Yaskawa INFORM job: OK_R2_O22-23(-90,180)OKKR.JBI

/JOB
//NAME OK_R2_O22-23(-90,180)OKKR
///FOLDERNAME X4
//POS
///NPOS 107,107,107,5,0,0
///TOOL 0
///POSTYPE PULSE
///PULSE
C00000=-79400,-96450,-73119,-47071,38510,50576
C00001=-120689,-37236,-43262,-1430,36977,65337
C00002=-120661,8390,6118,-1752,30038,65509
C00003=-121363,14227,14389,-901,27936,65072
C00004=-121630,18134,20803,-569,25994,64899
C00005=-122051,20456,22985,52,25844,64579
C00006=-122335,22651,22887,-209,31352,64420
C00007=-122335,23153,24532,-213,30597,64422
C00008=-122573,22007,22272,73,31399,64269
C00009=-118553,33336,34533,32200,31167,63632
C00010=-118554,33797,35647,32601,30785,63423
C00011=-118795,35881,37778,33055,30674,63177
C00012=-119029,34698,36884,33342,30719,63021
C00013=-119029,35470,39068,34241,29924,62556
C00014=-119029,34698,36884,33342,30719,63021
C00015=-122566,16275,19454,818,25870,64189
C00016=-120682,5973,-10666,26006,48512,34380
C00017=-120682,6077,-8041,26626,47105,33962
C00018=-120965,19546,-3322,22995,60520,37308
C00019=-120686,6056,-8291,26571,47234,33999
C00020=-120521,4024,-8795,26757,46523,33864
C00021=-122243,21545,4650,37838,56763,29509
C00022=-115724,34900,14421,35017,60862,31707
C00023=-122685,12952,-4874,39297,55027,28576
C00024=-131885,-4518,-22891,42927,60902,26587
C00025=-120689,-37236,-43262,-1430,36977,65337
C00026=-79400,-96450,-73119,-47071,38510,50576
C00027=8645,-72931,-67050,-57733,95594,74029
C00028=3643,-76224,-106676,19950,71810,76872
C00029=266,-73751,-67438,-57600,90404,72524
C00030=-56065,-40103,-98025,-15235,73272,62938
C00031=-80290,13979,-35130,-8518,69424,54762
C00032=-81621,16186,-30024,-7817,67316,54480
C00033=-82138,17140,-27919,-7543,66474,54366
C00034=-82701,19213,-25983,-7203,66302,54190
C00035=-82138,17140,-27919,-7543,66474,54366
C00036=-82074,13923,-28800,-7646,65378,54460
C00037=-82073,13446,-28104,-7686,64710,54504
C00038=-82074,14344,-29367,-7613,65938,54423
C00039=-80200,10192,-35655,-8662,67827,54907
C00040=-80279,11679,-32768,-3860,64531,54120
C00041=-80277,10318,-30958,-3920,62722,54182
C00042=-80747,9882,-30077,-3637,61936,54046
C00043=-80280,10347,-31011,-3916,62769,54180
C00044=-79691,8209,-31623,-4330,62077,54408
C00045=-80388,10283,-29809,-3872,61992,54168
C00046=-75315,21698,-19319,-7250,61724,55953
C00047=-80303,10454,-30913,-3901,62763,54172
C00048=-80304,11819,-32719,-3842,64572,54110
C00049=-56065,-40103,-98025,-15235,73272,62938
C00050=3643,-76224,-106676,19950,71810,76872
C00051=266,-73751,-67438,-57600,90404,72524
C00052=266,-73751,-67438,-57600,90404,72524
C00053=266,-73751,-67438,-57600,90404,72524
C00054=266,-73751,-67438,-57600,90404,72524
C00055=266,-73751,-67438,-57600,90404,72524
C00056=266,-73751,-67438,-57600,90404,72524
C00057=266,-73751,-67438,-57600,90404,72524
C00058=266,-73751,-67438,-57600,90404,72524
C00059=266,-73751,-67438,-57600,90404,72524
C00060=-120677,-3480,-20614,-18181,54095,-39471
C00061=-120311,11594,-4773,-18885,52273,-38972
C00062=-120169,13967,1466,-19666,49827,-38417
C00063=-119883,15460,2829,-19877,49828,-38285
C00064=-119880,14569,2014,-19868,49870,-38293
C00065=-119880,14692,3030,-20029,49339,-38180
C00066=-119880,15002,5218,-20385,48223,-37938
C00067=-119880,14692,3030,-20029,49339,-38180
C00068=-121128,7117,-4698,-18949,49860,-38864
C00069=-120984,8550,-10493,-36755,60982,-29079
C00070=-120492,10444,-8592,-38530,61785,-27976
C00071=-119910,12056,-7149,-38807,61994,-27785
C00072=-120247,11117,-7991,-38646,61874,-27896
C00073=-120247,11130,-6123,-39024,60976,-27528
C00074=-120247,11117,-7991,-38646,61874,-27896
C00075=-118757,6782,-7537,-20091,51910,-38210
C00076=-120681,6612,-10378,-25984,47448,-35852
C00077=-120681,6707,-7755,-26629,46038,-35426
C00078=-120905,15953,-5134,-22230,56700,-38204
C00079=-120839,4648,-8519,-26766,45460,-35327
C00080=-120685,6692,-7997,-26566,46163,-35467
C00081=-117777,13176,-6800,-24861,56252,-36867
C00082=-124527,9710,-9382,-30545,58873,-31634
C00083=-123617,18824,-2123,-35553,64566,-29659
C00084=-120681,6624,-6675,-42630,54896,-24176
C00085=-115739,6767,-11022,-43739,59328,-23743
C00086=266,-73751,-67438,-57600,90404,72524
C00087=266,-73751,-67438,-57600,90404,72524
C00088=-73074,14271,-65905,-40005,100084,-34925
C00089=-80386,15191,-35510,-35923,83035,-31364
C00090=-81077,18148,-29671,-35761,81084,-30977
C00091=-80079,11495,-28631,-39585,73800,-28709
C00092=-80398,13741,-26603,-39455,73592,-28760
C00093=-80079,11495,-28631,-39585,73800,-28709
C00094=-81415,17339,-25976,-35859,78754,-30337
C00095=-81415,16938,-25408,-35919,78297,-30186
C00096=-80477,16259,-27610,-36210,79478,-30223
C00097=-80390,10982,-30842,-41019,80930,-29700
C00098=-75383,13683,-22290,-51121,80669,-25817
C00099=-80082,8484,-31856,-41199,80558,-29427
C00100=-80393,11011,-30897,-41013,80966,-29715
C00101=-75635,11666,-22596,-52724,79323,-24782
C00102=-81650,7127,-27228,-49906,76991,-26356
C00103=-81866,7848,-27047,-49551,77560,-26716
C00104=-80364,10836,-30874,-41034,80899,-29677
C00105=-80366,12212,-32666,-40889,82284,-30221
C00106=-73074,14271,-65905,-40005,100084,-34925
BC00000=125925,693938,117612
BC00001=160005,693938,117612
BC00002=160005,693938,117612
BC00003=160005,693938,117612
BC00004=160005,693938,117612
BC00005=160005,693938,117612
BC00006=160005,693938,117612
BC00007=160005,693938,117612
BC00008=160005,693938,117612
BC00009=160005,693938,117612
BC00010=160005,693938,117612
BC00011=160005,693938,117612
BC00012=160005,693938,117612
BC00013=160005,693938,117612
BC00014=160005,693938,117612
BC00015=160005,693938,117612
BC00016=109874,700216,53
BC00017=109468,706283,53
BC00018=109365,707824,53
BC00019=109305,708710,53
BC00020=109305,708710,53
BC00021=161928,716448,53
BC00022=161928,716448,53
BC00023=161928,716448,53
BC00024=161928,716448,53
BC00025=160005,693938,117612
BC00026=125925,693938,117612
BC00027=97174,679874,426359
BC00028=199464,674570,1075173
BC00029=97174,666880,1005640
BC00030=48447,721710,1061717
BC00031=36753,734869,1075175
BC00032=36753,734869,1075175
BC00033=36753,734869,1075175
BC00034=36753,734869,1075175
BC00035=36753,734869,1075175
BC00036=36753,734869,1075175
BC00037=36753,734869,1075175
BC00038=36753,734869,1075175
BC00039=36753,734869,1075175
BC00040=22779,736990,1075175
BC00041=22483,742436,1075175
BC00042=22365,744614,1075175
BC00043=22365,744614,1075175
BC00044=22365,744614,1075175
BC00045=64164,751883,1075175
BC00046=64164,751883,1075175
BC00047=64283,749705,1075175
BC00048=64578,744259,1075175
BC00049=48447,721710,1061717
BC00050=199464,674570,1075173
BC00051=97174,666880,1005640
BC00052=97174,666880,922210
BC00053=97174,666880,922210
BC00054=97174,666880,918604
BC00055=97174,666880,720089
BC00056=97174,666880,697617
BC00057=97174,666880,697617
BC00058=97174,666880,426359
BC00059=97174,666880,426359
BC00060=311356,706634,69323
BC00061=311356,706634,69323
BC00062=311356,706634,69323
BC00063=311356,706634,69323
BC00064=311356,706634,69323
BC00065=311356,706634,69323
BC00066=311356,706634,69323
BC00067=311356,706634,69323
BC00068=311356,706634,69323
BC00069=275687,731318,6455
BC00070=272447,733560,745
BC00071=272447,733560,745
BC00072=272447,733560,745
BC00073=272447,733560,745
BC00074=272447,733560,745
BC00075=311356,706634,69323
BC00076=328879,699206,53
BC00077=329318,705264,53
BC00078=329461,707239,53
BC00079=329494,707688,53
BC00080=329494,707688,53
BC00081=268725,718156,53
BC00082=272132,734200,53
BC00083=272132,734200,53
BC00084=272781,731773,53
BC00085=274403,725707,53
BC00086=97174,666880,426359
BC00087=97174,666880,1033213
BC00088=194082,683690,1075175
BC00089=194082,735853,1075175
BC00090=194082,735853,1075175
BC00091=194082,735853,1075175
BC00092=194082,735853,1075175
BC00093=194082,735853,1075175
BC00094=194082,735853,1075175
BC00095=194082,735853,1075175
BC00096=194082,735853,1075175
BC00097=207750,742978,1075175
BC00098=207882,745158,1075175
BC00099=207882,745158,1075175
BC00100=207882,745158,1075175
BC00101=170775,751555,1075175
BC00102=170775,751555,1075175
BC00103=170775,751555,1075175
BC00104=165937,750176,1075175
BC00105=165607,744726,1075175
BC00106=194082,683690,1075175
EC00000=-798156,1112951
EC00001=-798156,1112951
EC00002=-798156,1112951
EC00003=-798156,1112951
EC00004=-798156,1112951
EC00005=-798156,1112951
EC00006=-798156,1112951
EC00007=-798156,1112951
EC00008=-798156,1112951
EC00009=-798156,1112951
EC00010=-798156,1112951
EC00011=-798156,1112951
EC00012=-798156,1112951
EC00013=-798156,1112951
EC00014=-798156,1112951
EC00015=-798156,1112951
EC00016=-798156,1112951
EC00017=-798156,1112951
EC00018=-798156,1112951
EC00019=-798156,1112951
EC00020=-798156,1112951
EC00021=-798156,1112951
EC00022=-798156,1112951
EC00023=-798156,1112951
EC00024=-798156,1112951
EC00025=-798156,1112951
EC00026=-798156,1112951
EC00027=-798156,1112951
EC00028=-798156,1112951
EC00029=-798156,1112951
EC00030=-798156,1112951
EC00031=-798156,1112951
EC00032=-798156,1112951
EC00033=-798156,1112951
EC00034=-798156,1112951
EC00035=-798156,1112951
EC00036=-798156,1112951
EC00037=-798156,1112951
EC00038=-798156,1112951
EC00039=-798156,1112951
EC00040=-798156,1112951
EC00041=-798156,1112951
EC00042=-798156,1112951
EC00043=-798156,1112951
EC00044=-798156,1112951
EC00045=-798156,1112951
EC00046=-798156,1112951
EC00047=-798156,1112951
EC00048=-798156,1112951
EC00049=-798156,1112951
EC00050=-798156,1112951
EC00051=-798156,1112951
EC00052=-861922,952659
EC00053=-880722,814928
EC00054=-879279,703703
EC00055=-885682,417967
EC00056=-877307,343621
EC00057=-877307,239254
EC00058=-798156,0
EC00059=-798156,0
EC00060=-798156,0
EC00061=-798156,0
EC00062=-798156,0
EC00063=-798156,0
EC00064=-798156,0
EC00065=-798156,0
EC00066=-798156,0
EC00067=-798156,0
EC00068=-798156,0
EC00069=-798156,0
EC00070=-798156,0
EC00071=-798156,0
EC00072=-798156,0
EC00073=-798156,0
EC00074=-798156,0
EC00075=-798156,0
EC00076=-798156,0
EC00077=-798156,0
EC00078=-798156,0
EC00079=-798156,0
EC00080=-798156,0
EC00081=-798156,0
EC00082=-798156,0
EC00083=-798156,0
EC00084=-798156,0
EC00085=-798156,0
EC00086=-798156,0
EC00087=-798156,0
EC00088=-798156,0
EC00089=-798156,0
EC00090=-798156,0
EC00091=-798156,0
EC00092=-798156,0
EC00093=-798156,0
EC00094=-798156,0
EC00095=-798156,0
EC00096=-798156,0
EC00097=-798156,0
EC00098=-798156,0
EC00099=-798156,0
EC00100=-798156,0
EC00101=-798156,0
EC00102=-798156,0
EC00103=-798156,0
EC00104=-798156,0
EC00105=-798156,0
EC00106=-798156,0
///POSTYPE BASE
///RECTAN
///RCONF 0,0,0,0,0,0,0,0,0,0,0,0,0,0,0,0,0,0,0,0,0,0,0,0
P00006=0.222,-3.123,-1.508,0.0000,0.0000,0.0000
P00021=-0.225,-6.128,-0.405,0.0000,0.0000,0.0000
P00022=0.222,-3.123,-1.508,0.0000,0.0000,0.0000
P00023=0.143,-0.036,0.682,0.0000,0.0000,0.0000
P00024=0.145,-0.552,1.326,0.0000,0.0000,0.0000
//INST
///DATE 2024/04/13 10:46
///ATTR SC,RW
///GROUP1 RB1,BS1
///GROUP2 ST1
NOP
'OK_r2_O22-23(-90,180)
MOVJ C00000 BC00000 VJ=100.00  +MOVJ EC00000 VJ=100.00
MOVJ C00001 BC00001 VJ=100.00  +MOVJ EC00001 VJ=100.00
'Path S1012
SFTOF3D
MOVJ C00002 BC00002 VJ=100.00  +MOVJ EC00002 VJ=100.00
MOVL C00003 BC00003 V=400.0  +MOVJ EC00003 VJ=100.00
SMOVL C00004 BC00004 V=133.3  +MOVJ EC00004
SREFP 3 C00005 BC00005  +REFP EC00005
CALL JOB:SEARCH-R1-S13D
SET P023 P006
SFTON3D P023
SMOVL C00006 BC00006 V=133.3  +MOVJ EC00006
SREFP 3 C00007 BC00007  +REFP EC00007
CALL JOB:SEARCH-R1-S13D
SET P023 P006
SFTON3D P023
SMOVL C00008 BC00008 V=166.7  +MOVJ EC00008
SFTOF3D
SMOVL C00009 BC00009 V=416.7  +MOVJ EC00009
SMOVL C00010 BC00010 V=166.7  +MOVJ EC00010
SREFP 3 C00011 BC00011  +REFP EC00011
CALL JOB:SEARCH-R1-S13D
SET P024 P006
SFTON3D P024
SMOVL C00012 BC00012 V=133.3  +MOVJ EC00012
SREFP 3 C00013 BC00013  +REFP EC00013
CALL JOB:SEARCH-R1-S13D
SET P024 P006
SFTON3D P024
SMOVL C00014 BC00014 V=166.7  +MOVJ EC00014
SFTOF3D
MOVL C00015 BC00015 V=400.0  +MOVJ EC00015 VJ=100.00
'Path W1013
SFTOF3D
SFTON3D P023
MOVJ C00016 BC00016 VJ=100.00  +MOVJ EC00016 VJ=100.00
SMOVL C00017 BC00017 V=400.0  +MOVJ EC00017
SMOVL C00018 BC00018 V=133.3 PL=0  +MOVJ EC00018
SREFP 1 C00019 BC00019  +REFP EC00019
SREFP 2 C00020 BC00020  +REFP EC00020
MACRO1 MJ#(0) ARGF6
ARCON
SFTON3D P024
SMOVL C00021 BC00021 V=7.5  +MOVJ EC00021
SMOVL C00022 BC00022 V=7.5  +MOVJ EC00022
ARCOF
SMOVL C00023 BC00023 V=400.0  +MOVJ EC00023
SMOVL C00024 BC00024 V=1000.0  +MOVJ EC00024
SFTOF3D
MOVJ C00025 BC00025 VJ=100.00  +MOVJ EC00025 VJ=100.00
MOVJ C00026 BC00026 VJ=100.00  +MOVJ EC00026 VJ=100.00
MOVJ C00027 BC00027 VJ=100.00  +MOVJ EC00027 VJ=100.00
'R-L Trip
MOVJ C00028 BC00028 VJ=100.00  +MOVJ EC00028 VJ=100.00
CALL JOB:CLEAN-R1_KM_NEW
MOVJ C00029 BC00029 VJ=100.00  +MOVJ EC00029 VJ=100.00
MOVJ C00030 BC00030 VJ=100.00  +MOVJ EC00030 VJ=100.00
'Path S1396
SFTOF3D
MOVJ C00031 BC00031 VJ=100.00  +MOVJ EC00031 VJ=100.00
MOVL C00032 BC00032 V=333.3  +MOVJ EC00032 VJ=100.00
SMOVL C00033 BC00033 V=166.7  +MOVJ EC00033
SREFP 3 C00034 BC00034  +REFP EC00034
CALL JOB:SEARCH-R1-S13D
SET P024 P006
SFTON3D P024
SMOVL C00035 BC00035 V=166.7  +MOVJ EC00035
SMOVL C00036 BC00036 V=166.7  +MOVJ EC00036
SREFP 3 C00037 BC00037  +REFP EC00037
CALL JOB:SEARCH-R1-S13D
SET P024 P006
SFTON3D P024
SMOVL C00038 BC00038 V=166.7  +MOVJ EC00038
MOVL C00039 BC00039 V=1000.0  +MOVJ EC00039 VJ=100.00
'Path W1397
SFTOF3D
SFTON3D P024
MOVJ C00040 BC00040 VJ=100.00  +MOVJ EC00040 VJ=100.00
SMOVL C00041 BC00041 V=400.0  +MOVJ EC00041
SMOVL C00042 BC00042 V=166.7 PL=0  +MOVJ EC00042
SREFP 1 C00043 BC00043  +REFP EC00043
SREFP 2 C00044 BC00044  +REFP EC00044
MACRO1 MJ#(0) ARGF6
ARCON
SMOVL C00045 BC00045 V=8.3  +MOVJ EC00045
SMOVL C00046 BC00046 V=8.3  +MOVJ EC00046
ARCOF
SMOVL C00047 BC00047 V=400.0  +MOVJ EC00047
SMOVL C00048 BC00048 V=1000.0  +MOVJ EC00048
SFTOF3D
MOVJ C00049 BC00049 VJ=100.00  +MOVJ EC00049 VJ=100.00
MOVJ C00050 BC00050 VJ=100.00  +MOVJ EC00050 VJ=100.00
CALL JOB:CLEAN-R1_KM_NEW
MOVJ C00051 BC00051 VJ=100.00  +MOVJ EC00051 VJ=100.00
MOVJ C00052 BC00052 VJ=100.00  +MOVJ EC00052 VJ=100.00
MOVJ C00053 BC00053 VJ=100.00  +MOVJ EC00053 VJ=100.00
MOVJ C00054 BC00054 VJ=100.00  +MOVJ EC00054 VJ=100.00
MOVJ C00055 BC00055 VJ=100.00  +MOVJ EC00055 VJ=100.00
MOVJ C00056 BC00056 VJ=100.00  +MOVJ EC00056 VJ=100.00
MOVJ C00057 BC00057 VJ=100.00  +MOVJ EC00057 VJ=100.00
MOVJ C00058 BC00058 VJ=100.00  +MOVJ EC00058 VJ=100.00
MOVJ C00059 BC00059 VJ=100.00  +MOVJ EC00059 VJ=100.00
'Path S1392
SFTOF3D
MOVJ C00060 BC00060 VJ=100.00  +MOVJ EC00060 VJ=100.00
MOVL C00061 BC00061 V=166.7  +MOVJ EC00061 VJ=100.00
SMOVL C00062 BC00062 V=166.7  +MOVJ EC00062
SREFP 3 C00063 BC00063  +REFP EC00063
CALL JOB:SEARCH-R1-S13D
SET P021 P006
SFTON3D P021
SMOVL C00064 BC00064 V=166.7  +MOVJ EC00064
SMOVL C00065 BC00065 V=166.7  +MOVJ EC00065
SREFP 3 C00066 BC00066  +REFP EC00066
CALL JOB:SEARCH-R1-S13D
SET P021 P006
SFTON3D P021
SMOVL C00067 BC00067 V=166.7  +MOVJ EC00067
SFTOF3D
MOVL C00068 BC00068 V=400.0  +MOVJ EC00068 VJ=100.00
SMOVL C00069 BC00069 V=666.7  +MOVJ EC00069
SMOVL C00070 BC00070 V=166.7  +MOVJ EC00070
SREFP 3 C00071 BC00071  +REFP EC00071
CALL JOB:SEARCH-R1-S13D
SET P022 P006
SFTON3D P022
SMOVL C00072 BC00072 V=166.7  +MOVJ EC00072
SREFP 3 C00073 BC00073  +REFP EC00073
CALL JOB:SEARCH-R1-S13D
SET P022 P006
SFTON3D P022
SMOVL C00074 BC00074 V=166.7  +MOVJ EC00074
MOVL C00075 BC00075 V=1000.0  +MOVJ EC00075 VJ=100.00
'Path W1393
SFTOF3D
SFTON3D P021
MOVJ C00076 BC00076 VJ=100.00  +MOVJ EC00076 VJ=100.00
SMOVL C00077 BC00077 V=400.0  +MOVJ EC00077
SMOVL C00078 BC00078 V=166.7 PL=0  +MOVJ EC00078
SREFP 1 C00079 BC00079  +REFP EC00079
SREFP 2 C00080 BC00080  +REFP EC00080
MACRO1 MJ#(0) ARGF6
ARCON
SFTON3D P022
SMOVL C00081 BC00081 V=7.5  +MOVJ EC00081
SMOVL C00082 BC00082 V=7.5  +MOVJ EC00082
SMOVL C00083 BC00083 V=7.5  +MOVJ EC00083
ARCOF
SFTOF3D
SMOVL C00084 BC00084 V=400.0  +MOVJ EC00084
SMOVL C00085 BC00085 V=1000.0  +MOVJ EC00085
SFTOF3D
'L-R Trip
MOVJ C00086 BC00086 VJ=100.00  +MOVJ EC00086 VJ=100.00
CALL JOB:CLEAN-R1_KM_NEW
MOVJ C00087 BC00087 VJ=100.00  +MOVJ EC00087 VJ=100.00
MOVJ C00088 BC00088 VJ=100.00  +MOVJ EC00088 VJ=100.00
'Path S1394
SFTOF3D
MOVJ C00089 BC00089 VJ=100.00  +MOVJ EC00089 VJ=100.00
MOVL C00090 BC00090 V=400.0  +MOVJ EC00090 VJ=100.00
SMOVL C00091 BC00091 V=166.7  +MOVJ EC00091
SREFP 3 C00092 BC00092  +REFP EC00092
CALL JOB:SEARCH-R1-S13D
SET P022 P006
SFTON3D P022
SMOVL C00093 BC00093 V=166.7  +MOVJ EC00093
SMOVL C00094 BC00094 V=166.7  +MOVJ EC00094
SREFP 3 C00095 BC00095  +REFP EC00095
CALL JOB:SEARCH-R1-S13D
SET P022 P006
SFTON3D P022
SMOVL C00096 BC00096 V=166.7  +MOVJ EC00096
'Path W1395
SFTOF3D
SFTON3D P022
SMOVL C00097 BC00097 V=400.0  +MOVJ EC00097
SMOVL C00098 BC00098 V=166.7 PL=0  +MOVJ EC00098
SREFP 1 C00099 BC00099  +REFP EC00099
SREFP 2 C00100 BC00100  +REFP EC00100
MACRO1 MJ#(0) ARGF6
ARCON
SMOVL C00101 BC00101 V=7.5  +MOVJ EC00101
SMOVL C00102 BC00102 V=7.5  +MOVJ EC00102
SMOVL C00103 BC00103 V=7.5  +MOVJ EC00103
ARCOF
SMOVL C00104 BC00104 V=400.0  +MOVJ EC00104
SMOVL C00105 BC00105 V=1000.0  +MOVJ EC00105
SFTOF3D
MOVJ C00106 BC00106 VJ=100.00  +MOVJ EC00106 VJ=100.00
END
